// TIA Portal V17 export
// export: Created 2023-02-13T11:16:22.2965313Z, ExportSetting WithDefaults, DisplayName Totally Integrated Automation Portal, DisplayVersion V17, DisplayName TIA Portal Openness, DisplayVersion V17, DisplayName TIA Portal Teamcenter Gateway, DisplayVersion V17, DisplayName TIA Portal Version Control Interface, DisplayVersion V17, DisplayName SINAMICS Startdrive Advanced, DisplayVersion V17, DisplayName SINAMICS Startdrive G130, G150, S120, S150, SINAMICS MV, S210, DisplayVersion V17, DisplayName SINAMICS Startdrive G110M, G120, G120C, G120D, G120P, G115D, DisplayVersion V17, DisplayName STEP 7 Professional, DisplayVersion V17, DisplayName STEP 7 Safety, DisplayVersion V17, DisplayName WinCC Professional, DisplayVersion V17
DATA_BLOCK "IO_Valve_Blend31_DB"   // DB61
VERSION : 0.1
// stored: AutoNumber true, DBAccessibleFromOPCUA true, DBAccessibleFromWebserver true, InstanceOfName IO_Valve_Blend31, InstanceOfType FB
"IO_Valve_Blend31"
   // VAR_INPUT
   //    "lock 1" : Bool;
   //    "lock 2" : Bool;
   //    "lock 3" : Bool;
   //    "lock 4" : Bool;
   //    init : Bool;
   //    reset : Bool;
   //    testing : Bool;
   // END_VAR
   // VAR
   //    "AV-31.01" : "Valve";
   //    "AV-31.02" : "Valve";
   //    "AV-31.03" : "Valve";
   //    "AV-31.04" : "Valve";
   //    "AV-31.05" : "Valve";
   //    "AV-31.06" : "Valve";
   //    "AV-31.07" : "Valve";
   //    "AV-31.08" : "Valve";
   //    "AV-31.09" : "Valve";
   //    "AV-31.10" : "Valve";
   //    "AV-31.11" : "Valve";
   //    "AV-31.21" : "Valve";
   //    "AV-31.22" : "Valve";
   //    "AV-31.23" : "Valve";
   //    "AV-31.24" : "Valve";
   //    "AV-31.25" : "Valve";
   //    "AV-31.26" : "Valve";
   //    "AV-31.27" : "Valve";
   //    "AV-31.28" : "Valve";
   //    "AV-31.29" : "Valve";
   //    "AV-31.30" : "Valve";
   //    "AV-31.31" : "Valve";
   //    "AV-31.32" : "Valve";
   //    "AV-31.33" : "Valve";
   //    "AV-31.34" : "Valve";
   //    "AV-31.35" : "Valve";
   //    "AV-31.41" : "Valve";
   //    "AV-31.42" : "Valve";
   // END_VAR
BEGIN
END_DATA_BLOCK
